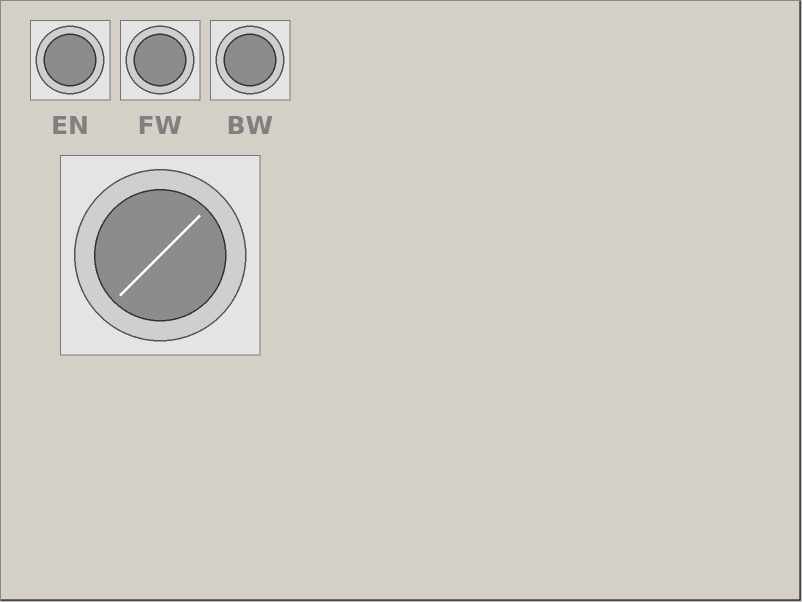
VISUALIZATION F02_Power  // 802x602
    Rectangle (0,0 800x600)
    Label (30,110 80x30), "EN"
    PushSwitchLed (30,20 80x80), variable: MAIN.axes[MAIN.hmiAxisSelect].bENABLE, behaviour: TOGGLE, style: Switch-PushSwitchLed-Gray
    PushSwitchLed (120,20 80x80), variable: MAIN.axes[MAIN.hmiAxisSelect].bEnFW, behaviour: TOGGLE, style: Switch-PushSwitchLed-Gray
    Label (120,110 80x30), "FW"
    PushSwitchLed (210,20 80x80), variable: MAIN.axes[MAIN.hmiAxisSelect].bEnBW, behaviour: TOGGLE, style: Switch-PushSwitchLed-Gray
    Label (210,110 80x30), "BW"
    Potentiometer360 (60,150 200x210), variable: MAIN.axes[MAIN.hmiAxisSelect].OVERRIDE, style: Potentiometer-Potentiometer360-Gray, scale format: %.1f, scale 0..100
        p2431819421: Outside
END_VISUALIZATION

(* stored: Version 1.1.0.1, ProductVersion 3.1.4022.7
   Visu F02_Power: Id {fdd2f889-e542-4bb7-99e9-d93103aed32a} *)
